// TIA Portal V16 export
// export: Created 2026-06-18T16:21:50.5636224Z, ExportSetting WithDefaults, DisplayName Totally Integrated Automation Portal, DisplayVersion V16 Update 8, DisplayName TIA Portal Version Control Interface, DisplayVersion V16 Update 8, DisplayName TIA Portal Openness, DisplayVersion V16 Update 8, DisplayName SINAMICS Startdrive Advanced, DisplayVersion V16, DisplayName SINAMICS Startdrive G130, G150, S120, S150, SINAMICS MV, S210, DisplayVersion V16, DisplayName SINAMICS Startdrive G110M, G120, G120C, G120D, G120P, DisplayVersion V16, DisplayName STEP 7 Professional, DisplayVersion V16 Update 8, DisplayName STEP 7 Safety, DisplayVersion V16 Update 7, DisplayName WinCC Advanced, DisplayVersion V16 Update 8
Screen "Login_Screen"  800x480, Number=1
  ScreenLayer 
    Circle "LMP_Online" at 250,388 size 48x48
    Button "BTN_Login" at 210,280 size 130x50  Mode=Text, TextOff="登录", TextOn="登录"
    Button "BTN_Logout" at 380,280 size 130x50  Mode=Text, TextOff="退出", TextOn="退出"
    IOField "IO_Username" at 270,120 size 220x40  DataFormat=Decimal, FormatPattern=9999999, Mode=InOutput
    IOField "IO_Password" at 270,190 size 220x40  DataFormat=Decimal, FormatPattern=9999999, Mode=InOutput
    SymbolicIOField "符号 I/O 域_1" at 457,258 size 96x32  CountVisibleItems=3, Mode=InOutput, OnValue=1, TextOff="0", TextOn="1"
    TextField "TXT_Title" at 200,30 size 400x44  Text="操作员登录"
    TextField "TXT_OnlineLabel" at 290,368 size 150x36  Text="在线状态"
    TextField "TXT_PasswordLabel" at 160,190 size 90x36  Text="密码"
    TextField "TXT_UserLabel" at 160,120 size 90x36  Text="用户名"
